// TIA Portal V21 export
TYPE "coneCrusherIOs"
   STRUCT
      luS : "lubricationSystemIOs";
      sg { S7_SetPoint := 'True'} : "switchgearInterface";
      self { S7_SetPoint := 'True'} : "coneCrusherInterface";
      btnStart : "LBC_typeDigitalSignalInterface";
      btnStop : "LBC_typeDigitalSignalInterface";
      keySwitch : "LBC_typeDigitalSignalInterface";
      emStop : "LBC_typeDigitalSignalInterface";
      btnReset : "LBC_typeDigitalSignalInterface";
      btnStartLuS : "LBC_typeDigitalSignalInterface";
      btnStopLuS : "LBC_typeDigitalSignalInterface";
      premoldingSw { S7_SetPoint := 'True'} : "LBC_typeDigitalSignalInterface";
      prestartAlmFb { S7_SetPoint := 'True'} : "LBC_typeDigitalSignalInterface";
      crusherEccentricTemp : "LBC_typeAnalogInputInterface";
      crusherOuterBearingTemp { S7_SetPoint := 'True'} : "LBC_typeAnalogInputInterface";
      crusherInnerBearingTemp { S7_SetPoint := 'True'} : "LBC_typeAnalogInputInterface";
      driveFrontBearingTemp { S7_SetPoint := 'True'} : "LBC_typeAnalogInputInterface";
      driveRearBearingTemp { S7_SetPoint := 'True'} : "LBC_typeAnalogInputInterface";
      driveWindingTempP1 { S7_SetPoint := 'True'} : "LBC_typeAnalogInputInterface";
      driveWindingTempP2 { S7_SetPoint := 'True'} : "LBC_typeAnalogInputInterface";
      driveWindingTempP3 { S7_SetPoint := 'True'} : "LBC_typeAnalogInputInterface";
      driveCurrent { S7_SetPoint := 'True'} : "LBC_typeAnalogInputInterface";
      sgReady { S7_SetPoint := 'True'} : "LBC_typeDigitalSignalInterface";
      sgFbOn { S7_SetPoint := 'True'} : "LBC_typeDigitalSignalInterface";
      sgFbOff { S7_SetPoint := 'True'} : "LBC_typeDigitalSignalInterface";
      sgStart : "LBC_typeDigitalSignalInterface";
      sgStop : "LBC_typeDigitalSignalInterface";
      preStartAlmOn : "LBC_typeDigitalSignalInterface";
      feedEn : "LBC_typeDigitalSignalInterface";   // Allow feed from upstream unit
   END_STRUCT;
END_TYPE
